      NOP   0;
// --- FCM 01 - Lifting devices ---
      L     "MAL1S032Par".Ilo.ILOMode;
      L     1;
      <>I   ;
      SPB   IO1;
// man on
      U     "MAL1S032Par".Ilo.GrCMDManOn[1];
      S     "G265M".Gr.InManual; // LIFTING DEVICE KILN 1
      R     "MAL1S032Par".Ilo.GrCMDManOn[1];
// man off
      U     "MAL1S032Par".Ilo.GrCMDManOff[1];
      S     "G265M".Gr.CmdManualOff; // LIFTING DEVICE KILN 1
      R     "G265M".Gr.InManual; // LIFTING DEVICE KILN 1
      R     "G265M".USW14; // ILO-cmd
      R     "G265M".USW15; // ILO-cmd
      R     "MAL1S032Par".Ilo.GrCMDManOff[1];
      R     "MAL1S032Par".Ilo.GrCMDManAdditional.Cmd1[1];
      R     "MAL1S032Par".Ilo.GrCMDManAdditional.Cmd2[1];
// man start
      U     "MAL1S032Par".Ilo.GrCMDManStart[1];
      S     "G265M".Gr.CmdOn; // LIFTING DEVICE KILN 1
      S     "G265M".Gr.CmdContinue; // LIFTING DEVICE KILN 1
      R     "MAL1S032Par".Ilo.GrCMDManStart[1];
      U     "MAL1S032Par".Ilo.GrCMDManStart[2];
      R     "MAL1S032Par".Ilo.GrCMDManStart[2];
// man stop
      U     "MAL1S032Par".Ilo.GrCMDManStop[1];
      S     "G265M".Gr.CmdOff; // LIFTING DEVICE KILN 1
      R     "MAL1S032Par".Ilo.GrCMDManStop[1];
// man fault reset
      U     "MAL1S032Par".Ilo.GrCMDManFaultReset[1];
      S     "G265M".Gr.CmdFaultReset; // LIFTING DEVICE KILN 1
      R     "MAL1S032Par".Ilo.GrCMDManFaultReset[1];
// moving direction
      UN    "G265M".Gr.InManual; // LIFTING DEVICE KILN 1
      O(    ;
      L     "MAL1S032Par".Ilo.Code_ILO_Funktion0;
      L     100;
      <>I   ;
      )     ;
      SPB   Stat;
      UN    "MAL1S032Par".Ilo.GrCMDManAdditional.Cmd1[1];
      UN    "MAL1S032Par".Ilo.GrCMDManAdditional.Cmd2[1];
      L     "MAL1S032Par".Par.MachineValue.SOLLWERT_HUBZUG1_HOEHE;
      SPB   Tpos;
      U     "MAL1S032Par".Ilo.GrCMDManAdditional.Cmd1[1]; // ManUp
      L     2000; // 1850mm + Offset = 2000mm
      SPB   Tpos;
      U     "MAL1S032Par".Ilo.GrCMDManAdditional.Cmd2[1]; // ManDown
      L     0; // 0mm
      SPB   Tpos;
      SPA   Stat;
// target position
Tpos: NOP   0;
      T     "MAL1S032Par".Par.ParIntProcess.TarPos_ILO_LiftDev;
Stat: NOP   0;
IO1:  NOP   0;
      NOP   0;
// --- FCM 04 - Fans ---
      L     "MAL1S032Par".Ilo.ILOMode;
      L     4;
      <>I   ;
      SPB   IO4;
// man on
      U     "MAL1S032Par".Ilo.GrCMDManOn[1];
      S     "G271M".Gr.InManual; // FAN KILN 1
//MW 2010.04.06
      S     "G273M".Gr.InManual; // RECYCLING AIR LOUVER KILN 1
      S     "G273M".Gr.CmdOn; // No Button: RECYCLING AIR LOUVER KILN 1
      S     "G273M".Gr.CmdContinue; // No Button RECYCLING AIR LOUVER KILN 1
      R     "MAL1S032Par".Ilo.GrCMDManOn[1];
// man off
      U     "MAL1S032Par".Ilo.GrCMDManOff[1];
      S     "G271M".Gr.CmdManualOff; // FAN KILN 1
      R     "G271M".Gr.InManual; // FAN KILN 1
      R     "G271M".USW14; // ILO-cmd
      R     "G271M".USW15; // ILO-cmd
//MW 2010.04.06
      S     "G273M".Gr.CmdManualOff; // RECYCLING AIR LOUVER KILN 1
      R     "G273M".Gr.InManual; // RECYCLING AIR LOUVER KILN 1
      R     "G273M".USW14; // ILO-cmd
      R     "G273M".USW15; // ILO-cmd
      R     "MAL1S032Par".Ilo.GrCMDManOff[1];
      R     "MAL1S032Par".Ilo.GrCMDManAdditional.Cmd1[1];
      R     "MAL1S032Par".Ilo.GrCMDManAdditional.Cmd2[1];
// man start
      U     "MAL1S032Par".Ilo.GrCMDManStart[1];
      S     "G271M".Gr.CmdOn; // FAN KILN 1
      S     "G271M".Gr.CmdContinue; // FAN KILN 1
//MW 2010.04.06
      S     "G273M".Gr.CmdOn; // No Button: RECYCLING AIR LOUVER KILN 1
      S     "G273M".Gr.CmdContinue; // No Button RECYCLING AIR LOUVER KILN 1
      R     "MAL1S032Par".Ilo.GrCMDManStart[1];
      U     "MAL1S032Par".Ilo.GrCMDManStart[2];
      R     "MAL1S032Par".Ilo.GrCMDManStart[2];
// man stop
      U     "MAL1S032Par".Ilo.GrCMDManStop[1];
      S     "G271M".Gr.CmdOff; // FAN KILN 1
//MW 2010.04.06
//      S     "G273M".Gr.CmdOff           // RECYCLING AIR LOUVER KILN 1
      R     "MAL1S032Par".Ilo.GrCMDManStop[1];
// man fault reset
      U     "MAL1S032Par".Ilo.GrCMDManFaultReset[1];
      S     "G271M".Gr.CmdFaultReset; // FAN KILN 1
//MW 2010.04.06
      S     "G273M".Gr.CmdFaultReset; // RECYCLING AIR LOUVER KILN 1
      R     "MAL1S032Par".Ilo.GrCMDManFaultReset[1];
// target position
      UN    "G271M".Gr.InManual; // FAN KILN 1
      O(    ;
      L     "MAL1S032Par".Ilo.Code_ILO_Funktion0;
      L     400;
      <>I   ;
      )     ;
      SPB   F04a;
      L     "MAL1S032Par".Ilo.SetpointInt01[1];
      T     "MAL1S032Par".Par.ParIntProcess.Speed_ILO_Fan;
F04a: NOP   0;
//MW 2010.04.06
      UN    "G273M".Gr.InManual; // Recycling Air Flap Kilningbox 1
      O(    ;
      L     "MAL1S032Par".Ilo.Code_ILO_Funktion0;
      L     400;
      <>I   ;
      )     ;
      SPB   F04b;
//MW      L     90                          // 90%
      L     100; // 100%
      T     "MAL1S032Par".Par.ParIntProcess.TarPos_ILO_RecycAir;
F04b: NOP   0;

IO4:  NOP   0;
      NOP   0;
// --- FCM 05 - Fans with target air temperature ---
      L     "MAL1S032Par".Ilo.ILOMode;
      L     5;
      <>I   ;
      SPB   IO5;
// man on
      U     "MAL1S032Par".Ilo.GrCMDManOn[1];
      S     "G271M".Gr.InManual; // FAN KILN 1
      S     "G273M".Gr.InManual; // RECYCLING AIR LOUVER KILN 1
      S     "G273M".Gr.CmdOn; // No Button: RECYCLING AIR LOUVER KILN 1
      S     "G273M".Gr.CmdContinue; // No Button RECYCLING AIR LOUVER KILN 1
      S     "G276M".Gr.InManual; // HEATING KILN 1
      S     "G276M".Gr.CmdOn; // No Button: HEATING KILN 1
      S     "G276M".Gr.CmdContinue; // No Button HEATING KILN 1
      S     "G277M".Gr.InManual; // LOUVER AIR HEATER 1 FOR KILN 1
      S     "G277M".Gr.CmdOn; // No Button: LOUVER AIR HEATER 1 FOR KILN 1
      S     "G277M".Gr.CmdContinue; // No Button LOUVER AIR HEATER 1 FOR KILN 1
//MW 2010.04.06      S     "G272M".Gr.InManual         // FRESH AIR LOUVER KILN 1
//MW 2010.04.06      S     "G272M".Gr.CmdOn            // No Button: FRESH AIR LOUVER KILN 1
//MW 2010.04.06      S     "G272M".Gr.CmdContinue      // No Button FRESH AIR LOUVER KILN 1
      S     "G278M".Gr.InManual; // WITHERING AIR KILN 1
      S     "G278M".Gr.CmdOn; // No Button: WITHERING AIR KILN 1
      S     "G278M".Gr.CmdContinue; // No Button WITHERING AIR KILN 1
      R     "MAL1S032Par".Ilo.GrCMDManOn[1];
// man off
      U     "MAL1S032Par".Ilo.GrCMDManOff[1];
      S     "G271M".Gr.CmdManualOff; // FAN KILN 1
      R     "G271M".Gr.InManual; // FAN KILN 1
      R     "G271M".USW14; // ILO-cmd
      R     "G271M".USW15; // ILO-cmd
      S     "G273M".Gr.CmdManualOff; // RECYCLING AIR LOUVER KILN 1
      R     "G273M".Gr.InManual; // RECYCLING AIR LOUVER KILN 1
      R     "G273M".USW14; // ILO-cmd
      R     "G273M".USW15; // ILO-cmd
      S     "G276M".Gr.CmdManualOff; // HEATING KILN 1
      R     "G276M".Gr.InManual; // HEATING KILN 1
      R     "G276M".USW14; // ILO-cmd
      R     "G276M".USW15; // ILO-cmd
      S     "G277M".Gr.CmdManualOff; // LOUVER AIR HEATER 1 FOR KILN 1
      R     "G277M".Gr.InManual; // LOUVER AIR HEATER 1 FOR KILN 1
      R     "G277M".USW14; // ILO-cmd
      R     "G277M".USW15; // ILO-cmd
//MW 2010.04.06      S     "G272M".Gr.CmdManualOff     // FRESH AIR LOUVER KILN 1
//MW 2010.04.06      R     "G272M".Gr.InManual         // FRESH AIR LOUVER KILN 1
      R     "G272M".USW14; // ILO-cmd
      R     "G272M".USW15; // ILO-cmd
      S     "G278M".Gr.CmdManualOff; // WITHERING AIR KILN 1
      R     "G278M".Gr.InManual; // WITHERING AIR KILN 1
      R     "G278M".USW14; // ILO-cmd
      R     "G278M".USW15; // ILO-cmd
      R     "MAL1S032Par".Ilo.GrCMDManOff[1];
      R     "MAL1S032Par".Ilo.GrCMDManAdditional.Cmd1[1];
      R     "MAL1S032Par".Ilo.GrCMDManAdditional.Cmd2[1];
// man start
      U     "MAL1S032Par".Ilo.GrCMDManStart[1];
      S     "G271M".Gr.CmdOn; // FAN KILN 1
      S     "G271M".Gr.CmdContinue; // FAN KILN 1
      S     "G273M".Gr.CmdOn; // RECYCLING AIR LOUVER KILN 1
      S     "G273M".Gr.CmdContinue; // RECYCLING AIR LOUVER KILN 1
      S     "G276M".Gr.CmdOn; // HEATING KILN 1
      S     "G276M".Gr.CmdContinue; // HEATING KILN 1
      S     "G277M".Gr.CmdOn; // LOUVER AIR HEATER 1 FOR KILN 1
      S     "G277M".Gr.CmdContinue; // LOUVER AIR HEATER 1 FOR KILN 1
//MW 2010.04.06      S     "G272M".Gr.CmdOn            // FRESH AIR LOUVER KILN 1
//MW 2010.04.06      S     "G272M".Gr.CmdContinue      // FRESH AIR LOUVER KILN 1
      S     "G278M".Gr.CmdOn; // WITHERING AIR KILN 1
      S     "G278M".Gr.CmdContinue; // WITHERING AIR KILN 1
      R     "MAL1S032Par".Ilo.GrCMDManStart[1];
      U     "MAL1S032Par".Ilo.GrCMDManStart[2];
      R     "MAL1S032Par".Ilo.GrCMDManStart[2];
// man stop
//MW 2010.04.14      U     "MAL1S032Par".Ilo.GrSTMan[17]
      U     "MAL1S032Par".Ilo.GrCMDManStop[1];
      S     "G271M".Gr.CmdOff; // FAN KILN 1
      S     "G273M".Gr.CmdOff; // RECYCLING AIR LOUVER KILN 1
      S     "G276M".Gr.CmdOff; // HEATING KILN 1
      S     "G277M".Gr.CmdOff; // LOUVER AIR HEATER 1 FOR KILN 1
//MW 2010.04.06      S     "G272M".Gr.CmdOff           // FRESH AIR LOUVER KILN 1
      S     "G278M".Gr.CmdOff; // WITHERING AIR KILN 1
//MW 2010.04.14      R     "MAL1S032Par".Ilo.GrSTMan[17]
      R     "MAL1S032Par".Ilo.GrCMDManStop[1];
// man fault reset
      U     "MAL1S032Par".Ilo.GrCMDManFaultReset[1];
      S     "G271M".Gr.CmdFaultReset; // FAN KILN 1
      S     "G273M".Gr.CmdFaultReset; // RECYCLING AIR LOUVER KILN 1
      S     "G276M".Gr.CmdFaultReset; // HEATING KILN 1
      S     "G277M".Gr.CmdFaultReset; // LOUVER AIR HEATER 1 FOR KILN 1
//MW 2010.04.06      S     "G272M".Gr.CmdFaultReset    // FRESH AIR LOUVER KILN 1
      S     "G278M".Gr.CmdFaultReset; // WITHERING AIR KILN 1
      R     "MAL1S032Par".Ilo.GrCMDManFaultReset[1];
// target position
      UN    "G271M".Gr.InManual; // FAN KILN 1
      O(    ;
      L     "MAL1S032Par".Ilo.Code_ILO_Funktion0;
      L     500;
      <>I   ;
      )     ;
      SPB   F05b;
      L     "MAL1S032Par".Ilo.SetpointInt01[1];
      T     "MAL1S032Par".Par.ParIntProcess.Speed_ILO_Fan;
F05b: NOP   0;
      UN    "G273M".Gr.InManual; // Recycling Air Flap Kilningbox 1
      O(    ;
      L     "MAL1S032Par".Ilo.Code_ILO_Funktion0;
      L     500;
      <>I   ;
      )     ;
      SPB   F05c;
      L     "MAL1S032Par".Ilo.SetpointInt03[1];
      T     "MAL1S032Par".Par.ParIntProcess.TarPos_ILO_RecycAir;
F05c: NOP   0;
      UN    "G278M".Gr.InManual; // Withering Air Flap Kilningbox 1
      O(    ;
      L     "MAL1S032Par".Ilo.Code_ILO_Funktion0;
      L     500;
      <>I   ;
      )     ;
      SPB   F05d;
      L     "MAL1S032Par".Ilo.SetpointInt04[1];
      T     "MAL1S032Par".Par.ParIntProcess.TarPos_ILO_WitheringAir;
F05d: NOP   0;
      UN    "G276M".Gr.InManual; // Heating Kiln 1
      O(    ;
      L     "MAL1S032Par".Ilo.Code_ILO_Funktion0;
      L     500;
      <>I   ;
      )     ;
      SPB   F05e;
//MW 2010.04.06      L     "MAL1S032Par".Ilo.SetpointInt01[2]
      L     "MAL1S032Par".Ilo.SetpointInt02[1];
      T     "MAL1S032Par".Par.ParIntProcess.TargetTemperature_ILO;
F05e: NOP   0;

IO5:  NOP   0;
      NOP   0;
// --- FCM 06 - Fresh air flap ---
      L     "MAL1S032Par".Ilo.ILOMode;
      L     6;
      <>I   ;
      SPB   IO6;
// man on
      U     "MAL1S032Par".Ilo.GrCMDManOn[1];
      S     "G272M".Gr.InManual; // FRESH AIR LOUVER KILN 1
      R     "MAL1S032Par".Ilo.GrCMDManOn[1];
// man off
      U     "MAL1S032Par".Ilo.GrCMDManOff[1];
      S     "G272M".Gr.CmdManualOff; // FRESH AIR LOUVER KILN 1
      R     "G272M".Gr.InManual; // FRESH AIR LOUVER KILN 1
      R     "G272M".USW14; // ILO-cmd
      R     "G272M".USW15; // ILO-cmd
      R     "MAL1S032Par".Ilo.GrCMDManOff[1];
      R     "MAL1S032Par".Ilo.GrCMDManAdditional.Cmd1[1];
      R     "MAL1S032Par".Ilo.GrCMDManAdditional.Cmd2[1];
// man start
      U     "MAL1S032Par".Ilo.GrCMDManStart[1];
      S     "G272M".Gr.CmdOn; // FRESH AIR LOUVER KILN 1
      S     "G272M".Gr.CmdContinue; // FRESH AIR LOUVER KILN 1
      R     "MAL1S032Par".Ilo.GrCMDManStart[1];
      U     "MAL1S032Par".Ilo.GrCMDManStart[2];
      R     "MAL1S032Par".Ilo.GrCMDManStart[2];
// man stop
      U     "MAL1S032Par".Ilo.GrCMDManStop[1];
      S     "G272M".Gr.CmdOff; // FRESH AIR LOUVER KILN 1
      R     "MAL1S032Par".Ilo.GrCMDManStop[1];
// man fault reset
      U     "MAL1S032Par".Ilo.GrCMDManFaultReset[1];
      S     "G272M".Gr.CmdFaultReset; // FRESH AIR LOUVER KILN 1
      R     "MAL1S032Par".Ilo.GrCMDManFaultReset[1];
// moving direction

// target position
      UN    "G272M".Gr.InManual; // FRESH AIR LOUVER KILN 1
      SPB   F06b;
      L     "MAL1S032Par".Ilo.SetpointInt01[1];
      T     "MAL1S032Par".Par.ParIntProcess.TarPos_ILO_FreshAir;
F06b: NOP   0;

IO6:  NOP   0;
      NOP   0;
// --- FCM 07 - Recycling air flap ---
      L     "MAL1S032Par".Ilo.ILOMode;
      L     7;
      <>I   ;
      SPB   IO7;
// man on
      U     "MAL1S032Par".Ilo.GrCMDManOn[1];
      S     "G273M".Gr.InManual; // RECYCLING AIR LOUVER KILN 1
      S     "G278M".Gr.InManual; // WITHERING AIR KILN 1
      R     "MAL1S032Par".Ilo.GrCMDManOn[1];
// man off
      U     "MAL1S032Par".Ilo.GrCMDManOff[1];
      S     "G273M".Gr.CmdManualOff; // RECYCLING AIR LOUVER KILN 1
      R     "G273M".Gr.InManual; // RECYCLING AIR LOUVER KILN 1
      R     "G273M".USW14; // ILO-cmd
      R     "G273M".USW15; // ILO-cmd
      S     "G278M".Gr.CmdManualOff; // WITHERING AIR KILN 1
      R     "G278M".Gr.InManual; // WITHERING AIR KILN 1
      R     "G278M".USW14; // ILO-cmd
      R     "G278M".USW15; // ILO-cmd
      R     "MAL1S032Par".Ilo.GrCMDManOff[1];
      R     "MAL1S032Par".Ilo.GrCMDManAdditional.Cmd1[1];
      R     "MAL1S032Par".Ilo.GrCMDManAdditional.Cmd2[1];
// man start
      U     "MAL1S032Par".Ilo.GrCMDManStart[1];
      S     "G273M".Gr.CmdOn; // RECYCLING AIR LOUVER KILN 1
      S     "G273M".Gr.CmdContinue; // RECYCLING AIR LOUVER KILN 1
      S     "G278M".Gr.CmdOn; // WITHERING AIR KILN 1
      S     "G278M".Gr.CmdContinue; // WITHERING AIR KILN 1
      R     "MAL1S032Par".Ilo.GrCMDManStart[1];
      U     "MAL1S032Par".Ilo.GrCMDManStart[2];
      R     "MAL1S032Par".Ilo.GrCMDManStart[2];
// man stop
      U     "MAL1S032Par".Ilo.GrCMDManStop[1];
      S     "G273M".Gr.CmdOff; // RECYCLING AIR LOUVER KILN 1
      S     "G278M".Gr.CmdOff; // WITHERING AIR KILN 1
      R     "MAL1S032Par".Ilo.GrCMDManStop[1];
// man fault reset
      U     "MAL1S032Par".Ilo.GrCMDManFaultReset[1];
      S     "G273M".Gr.CmdFaultReset; // RECYCLING AIR LOUVER KILN 1
      S     "G278M".Gr.CmdFaultReset; // WITHERING AIR KILN 1
      R     "MAL1S032Par".Ilo.GrCMDManFaultReset[1];
// moving direction

// target position
      UN    "G273M".Gr.InManual; // RECYCLING AIR LOUVER KILN 1
      SPB   F07a;
      L     "MAL1S032Par".Ilo.SetpointInt01[1];
      T     "MAL1S032Par".Par.ParIntProcess.TarPos_ILO_RecycAir;
F07a: NOP   0;
IO7:  NOP   0;
      NOP   0;
// --- FCM 09 - Floor drives ---
      L     "MAL1S032Par".Ilo.ILOMode;
      L     9;
      <>I   ;
      SPB   IO9;
// man on
      U     "MAL1S032Par".Ilo.GrCMDManOn[1];
      S     "G266M".Gr.InManual; // TRAVELLING DRIVE KILN 1
      R     "MAL1S032Par".Ilo.GrCMDManOn[1];
// man off
      U     "MAL1S032Par".Ilo.GrCMDManOff[1];
      S     "G266M".Gr.CmdManualOff; // TRAVELLING DRIVE KILN 1
      R     "G266M".Gr.InManual; // TRAVELLING DRIVE KILN 1
      R     "G266M".USW14; // ILO-cmd
      R     "G266M".USW15; // ILO-cmd
      R     "MAL1S032Par".Ilo.GrCMDManOff[1];
      R     "MAL1S032Par".Ilo.GrCMDManAdditional.Cmd1[1];
      R     "MAL1S032Par".Ilo.GrCMDManAdditional.Cmd2[1];
// man start
      U     "MAL1S032Par".Ilo.GrCMDManStart[1];
      S     "G266M".Gr.CmdOn; // TRAVELLING DRIVE KILN 1
      S     "G266M".Gr.CmdContinue; // TRAVELLING DRIVE KILN 1
      R     "MAL1S032Par".Ilo.GrCMDManStart[1];
      U     "MAL1S032Par".Ilo.GrCMDManStart[2];
      R     "MAL1S032Par".Ilo.GrCMDManStart[2];
// man stop
      U     "MAL1S032Par".Ilo.GrCMDManStop[1];
      S     "G266M".Gr.CmdOff; // TRAVELLING DRIVE KILN 1
      R     "MAL1S032Par".Ilo.GrCMDManStop[1];
// man fault reset
      U     "MAL1S032Par".Ilo.GrCMDManFaultReset[1];
      S     "G266M".Gr.CmdFaultReset; // TRAVELLING DRIVE KILN 1
      R     "MAL1S032Par".Ilo.GrCMDManFaultReset[1];
      NOP   0;
      UN    "G266M".Gr.InManual; // TRAVELLING DRIVE KILN 1
      O     ;
      UN    "MAL1S032Par".Ilo.GrCMDManAdditional.Cmd1[1];
      UN    "MAL1S032Par".Ilo.GrCMDManAdditional.Cmd2[1];
      SPB   f092;
      U     "MAL1S032Par".Ilo.GrCMDManAdditional.Cmd1[1];
      =     "G266M".USW14; // ILO-cmd run fwd
      U     "MAL1S032Par".Ilo.GrCMDManAdditional.Cmd2[1];
      =     "G266M".USW15; // ILO-cmd run rev
// target position
      L     "MAL1S032Par".Ilo.SetpointInt01[1];
      T     "MAL1S032Par".Par.ParIntProcess.Speed_ILO_FloorRotating;
f092: NOP   0;

IO9:  NOP   0;
      NOP   0;
// --- FCM 10 - Floor drives and lifting devices ---
      L     "MAL1S032Par".Ilo.ILOMode;
      L     10;
      <>I   ;
      SPB   IO10;
// man on
      U     "MAL1S032Par".Ilo.GrCMDManOn[1];
      S     "G265M".Gr.InManual; // LIFTING DEVICE KILN 1
      S     "G265M".Gr.CmdOn; // No Button: LIFTING DEVICE KILN 1
      S     "G265M".Gr.CmdContinue; // No Button LIFTING DEVICE KILN 1
      S     "G266M".Gr.InManual; // TRAVELLING DRIVE KILN 1
      R     "MAL1S032Par".Ilo.GrCMDManOn[1];
// man off
      U     "MAL1S032Par".Ilo.GrCMDManOff[1];
      S     "G265M".Gr.CmdManualOff; // LIFTING DEVICE KILN 1
      R     "G265M".Gr.InManual; // LIFTING DEVICE KILN 1
      R     "G265M".USW14; // ILO-cmd
      R     "G265M".USW15; // ILO-cmd
      S     "G266M".Gr.CmdManualOff; // TRAVELLING DRIVE KILN 1
      R     "G266M".Gr.InManual; // TRAVELLING DRIVE KILN 1
      R     "G266M".USW14; // ILO-cmd
      R     "G266M".USW15; // ILO-cmd
      R     "MAL1S032Par".Ilo.GrCMDManOff[1];
      R     "MAL1S032Par".Ilo.GrCMDManAdditional.Cmd1[1];
      R     "MAL1S032Par".Ilo.GrCMDManAdditional.Cmd2[1];
// man start
      U     "MAL1S032Par".Ilo.GrCMDManStart[1];
      S     "G266M".Gr.CmdOn; // TRAVELLING DRIVE KILN 1
      S     "G266M".Gr.CmdContinue; // TRAVELLING DRIVE KILN 1
      R     "MAL1S032Par".Ilo.GrCMDManStart[1];
      U     "MAL1S032Par".Ilo.GrCMDManStart[2];
      S     "G265M".Gr.CmdOn; // LIFTING DEVICE KILN 1
      S     "G265M".Gr.CmdContinue; // LIFTING DEVICE KILN 1
      R     "MAL1S032Par".Ilo.GrCMDManStart[2];
      U     "MAL1S032Par".Ilo.GrCMDManStart[3];
      R     "MAL1S032Par".Ilo.GrCMDManStart[3];
// man stop
      U     "MAL1S032Par".Ilo.GrCMDManStop[1];
      S     "G265M".Gr.CmdOff; // LIFTING DEVICE KILN 1
      S     "G266M".Gr.CmdOff; // TRAVELLING DRIVE KILN 1
      R     "MAL1S032Par".Ilo.GrCMDManStop[1];
// man fault reset
      U     "MAL1S032Par".Ilo.GrCMDManFaultReset[1];
      S     "G265M".Gr.CmdFaultReset; // LIFTING DEVICE KILN 1
      S     "G266M".Gr.CmdFaultReset; // TRAVELLING DRIVE KILN 1
      R     "MAL1S032Par".Ilo.GrCMDManFaultReset[1];
// moving direction
      NOP   0;
      UN    "G266M".Gr.InManual; // TRAVELLING DRIVE KILN 1
      O     ;
      UN    "MAL1S032Par".Ilo.GrCMDManAdditional.Cmd1[1];
      UN    "MAL1S032Par".Ilo.GrCMDManAdditional.Cmd2[1];
      SPB   f102;
      U     "MAL1S032Par".Ilo.GrCMDManAdditional.Cmd1[1];
      =     "G266M".USW14; // ILO-cmd run fwd
      U     "MAL1S032Par".Ilo.GrCMDManAdditional.Cmd2[1];
      =     "G266M".USW15; // ILO-cmd run rev
// target speed floor drives
      L     "MAL1S032Par".Ilo.SetpointInt01[1];
      T     "MAL1S032Par".Par.ParIntProcess.Speed_ILO_FloorRotating;
f102: NOP   0;
      UN    "G265M".Gr.InManual; // LIFTING DEVICE KILN 1
      O(    ;
      L     "MAL1S032Par".Ilo.Code_ILO_Funktion0;
      L     1000;
      <>I   ;
      )     ;
      SPB   f103;
// target position lifting devices
      L     "MAL1S032Par".Ilo.SetpointInt02[1];
      T     "MAL1S032Par".Par.ParIntProcess.TarPos_ILO_LiftDev;
f103: NOP   0;

IO10: NOP   0;
      NOP   0;
// --- FCM 11 - Floor drives and lifting devices and screw ---
      L     "MAL1S032Par".Ilo.ILOMode;
      L     11;
      <>I   ;
      SPB   IO11;
// man on
      U     "MAL1S032Par".Ilo.GrCMDManOn[1];
      S     "G265M".Gr.InManual; // LIFTING DEVICE KILN 1
      S     "G265M".Gr.CmdOn; // No Button: LIFTING DEVICE KILN 1
      S     "G265M".Gr.CmdContinue; // No Button LIFTING DEVICE KILN 1
      S     "G266M".Gr.InManual; // TRAVELLING DRIVE KILN 1
      S     "G267M".Gr.InManual; // UNLOADING / LOADING SCREW KILN 1
      R     "MAL1S032Par".Ilo.GrCMDManOn[1];
// man off
      U     "MAL1S032Par".Ilo.GrCMDManOff[1];
      S     "G265M".Gr.CmdManualOff; // LIFTING DEVICE KILN 1
      R     "G265M".Gr.InManual; // LIFTING DEVICE KILN 1
      R     "G265M".USW14; // ILO-cmd
      R     "G265M".USW15; // ILO-cmd
      S     "G266M".Gr.CmdManualOff; // TRAVELLING DRIVE KILN 1
      R     "G266M".Gr.InManual; // TRAVELLING DRIVE KILN 1
      R     "G266M".USW14; // ILO-cmd
      R     "G266M".USW15; // ILO-cmd
      S     "G267M".Gr.CmdManualOff; // UNLOADING / LOADING SCREW KILN 1
      R     "G267M".Gr.InManual; // UNLOADING / LOADING SCREW KILN 1
      R     "G267M".USW14; // ILO-cmd
      R     "G267M".USW15; // ILO-cmd
      R     "MAL1S032Par".Ilo.GrCMDManOff[1];
      R     "MAL1S032Par".Ilo.GrCMDManAdditional.Cmd1[1];
      R     "MAL1S032Par".Ilo.GrCMDManAdditional.Cmd2[1];
// man start
      U     "MAL1S032Par".Ilo.GrCMDManStart[1];
      S     "G266M".Gr.CmdOn; // TRAVELLING DRIVE KILN 1
      S     "G266M".Gr.CmdContinue; // TRAVELLING DRIVE KILN 1
      R     "MAL1S032Par".Ilo.GrCMDManStart[1];
      U     "MAL1S032Par".Ilo.GrCMDManStart[2];
      S     "G265M".Gr.CmdOn; // LIFTING DEVICE KILN 1
      S     "G265M".Gr.CmdContinue; // LIFTING DEVICE KILN 1
      R     "MAL1S032Par".Ilo.GrCMDManStart[2];
      U     "MAL1S032Par".Ilo.GrCMDManStart[3];
      S     "G267M".Gr.CmdOn; // UNLOADING / LOADING SCREW KILN 1
      S     "G267M".Gr.CmdContinue; // UNLOADING / LOADING SCREW KILN 1
      R     "MAL1S032Par".Ilo.GrCMDManStart[3];
//MW      U     "MAL1S032Par".Ilo.GrCMDManStart[4]
//MW      S     "G267M".Gr.CmdOn            // UNLOADING / LOADING SCREW KILN 1
//MW      S     "G267M".Gr.CmdContinue      // UNLOADING / LOADING SCREW KILN 1
//MW      R     "MAL1S032Par".Ilo.GrCMDManStart[4]
// man stop
      U     "MAL1S032Par".Ilo.GrCMDManStop[1];
      S     "G265M".Gr.CmdOff; // LIFTING DEVICE KILN 1
      S     "G266M".Gr.CmdOff; // TRAVELLING DRIVE KILN 1
      S     "G267M".Gr.CmdOff; // UNLOADING / LOADING SCREW KILN 1
      R     "MAL1S032Par".Ilo.GrCMDManStop[1];
// man fault reset
      U     "MAL1S032Par".Ilo.GrCMDManFaultReset[1];
      S     "G265M".Gr.CmdFaultReset; // LIFTING DEVICE KILN 1
      S     "G266M".Gr.CmdFaultReset; // TRAVELLING DRIVE KILN 1
      S     "G267M".Gr.CmdFaultReset; // UNLOADING / LOADING SCREW KILN 1
      R     "MAL1S032Par".Ilo.GrCMDManFaultReset[1];
// moving direction
      UN    "G266M".Gr.InManual; // TRAVELLING DRIVE KILN 1
      O     ;
      UN    "MAL1S032Par".Ilo.GrCMDManAdditional.Cmd1[1];
      UN    "MAL1S032Par".Ilo.GrCMDManAdditional.Cmd2[1];
      SPB   f112;
      U     "MAL1S032Par".Ilo.GrCMDManAdditional.Cmd1[1];
      =     "G266M".USW14; // ILO-cmd run fwd
      U     "MAL1S032Par".Ilo.GrCMDManAdditional.Cmd2[1];
      =     "G266M".USW15; // ILO-cmd run rev
// target speed floor drives
      L     "MAL1S032Par".Ilo.SetpointInt01[1];
      T     "MAL1S032Par".Par.ParIntProcess.Speed_ILO_FloorRotating;
f112: NOP   0;
      UN    "G265M".Gr.InManual; // Malting Plant OAO Belsolod Ivanonvo Weissrussland
      O(    ;
      L     "MAL1S032Par".Ilo.Code_ILO_Funktion0;
      L     1100;
      <>I   ;
      )     ;
      SPB   f113;
// target position lifting devices
      L     "MAL1S032Par".Ilo.SetpointInt01[2];
      L     "MAL1S032Par".Ilo.SetpointInt02[1];
      T     "MAL1S032Par".Par.ParIntProcess.TarPos_ILO_LiftDev;
f113: NOP   0;
      UN    "G267M".Gr.InManual; // UNLOADING / LOADING SCREW KILN 1
      O     ;
      UN    "MAL1S032Par".Ilo.GrCMDManAdditional.Cmd1[3];
      UN    "MAL1S032Par".Ilo.GrCMDManAdditional.Cmd2[3];
      SPB   f114;
      U     "MAL1S032Par".Ilo.GrCMDManAdditional.Cmd1[3];
      =     "G267M".USW14; // ILO-cmd run fwd
      U     "MAL1S032Par".Ilo.GrCMDManAdditional.Cmd2[3];
      =     "G267M".USW15; // ILO-cmd run rev
f114: NOP   0;
IO11: NOP   0;
      NOP   0;
// --- FCM 12 - Floor drives and lifting devices and screw and discharging flap ---
      L     "MAL1S032Par".Ilo.ILOMode;
      L     12;
      <>I   ;
      SPB   IO12;
// man on
      U     "MAL1S032Par".Ilo.GrCMDManOn[1];
      S     "G265M".Gr.InManual; // LIFTING DEVICE KILN 1
      S     "G265M".Gr.CmdOn; // No Button: LIFTING DEVICE KILN 1
      S     "G265M".Gr.CmdContinue; // No Button LIFTING DEVICE KILN 1
      S     "G266M".Gr.InManual; // TRAVELLING DRIVE KILN 1
      S     "G267M".Gr.InManual; // UNLOADING / LOADING SCREW KILN 1
      S     "G268M".Gr.InManual; // DISCHARGE DOOR KILN 1
      R     "MAL1S032Par".Ilo.GrCMDManOn[1];
// man off
      U     "MAL1S032Par".Ilo.GrCMDManOff[1];
      S     "G265M".Gr.CmdManualOff; // LIFTING DEVICE KILN 1
      R     "G265M".Gr.InManual; // LIFTING DEVICE KILN 1
      R     "G265M".USW14; // ILO-cmd
      R     "G265M".USW15; // ILO-cmd
      S     "G266M".Gr.CmdManualOff; // TRAVELLING DRIVE KILN 1
      R     "G266M".Gr.InManual; // TRAVELLING DRIVE KILN 1
      R     "G266M".USW14; // ILO-cmd
      R     "G266M".USW15; // ILO-cmd
      S     "G267M".Gr.CmdManualOff; // UNLOADING / LOADING SCREW KILN 1
      R     "G267M".Gr.InManual; // UNLOADING / LOADING SCREW KILN 1
      R     "G267M".USW14; // ILO-cmd
      R     "G267M".USW15; // ILO-cmd
      S     "G268M".Gr.CmdManualOff; // DISCHARGE DOOR KILN 1
      R     "G268M".Gr.InManual; // DISCHARGE DOOR KILN 1
      R     "G268M".USW14; // ILO-cmd
      R     "G268M".USW15; // ILO-cmd
      R     "MAL1S032Par".Ilo.GrCMDManOff[1];
      R     "MAL1S032Par".Ilo.GrCMDManAdditional.Cmd1[1];
      R     "MAL1S032Par".Ilo.GrCMDManAdditional.Cmd2[1];
// man start
      U     "MAL1S032Par".Ilo.GrCMDManStart[1];
      S     "G266M".Gr.CmdOn; // TRAVELLING DRIVE KILN 1
      S     "G266M".Gr.CmdContinue; // TRAVELLING DRIVE KILN 1
      R     "MAL1S032Par".Ilo.GrCMDManStart[1];
      U     "MAL1S032Par".Ilo.GrCMDManStart[2];
      S     "G265M".Gr.CmdOn; // LIFTING DEVICE KILN 1
      S     "G265M".Gr.CmdContinue; // LIFTING DEVICE KILN 1
      R     "MAL1S032Par".Ilo.GrCMDManStart[2];
      U     "MAL1S032Par".Ilo.GrCMDManStart[3];
      S     "G267M".Gr.CmdOn; // UNLOADING / LOADING SCREW KILN 1
      S     "G267M".Gr.CmdContinue; // UNLOADING / LOADING SCREW KILN 1
      R     "MAL1S032Par".Ilo.GrCMDManStart[3];
      U     "MAL1S032Par".Ilo.GrCMDManStart[4];
//MW 2010.04.16      S     "G267M".Gr.CmdOn            // UNLOADING / LOADING SCREW KILN 1
//MW 2010.04.16      S     "G267M".Gr.CmdContinue      // UNLOADING / LOADING SCREW KILN 1
      S     "G268M".Gr.CmdOn; // DISCHARGE DOOR KILN 1
      S     "G268M".Gr.CmdContinue; // DISCHARGE DOOR KILN 1
      R     "MAL1S032Par".Ilo.GrCMDManStart[4];
// man stop
      U     "MAL1S032Par".Ilo.GrCMDManStop[1];
      S     "G265M".Gr.CmdOff; // LIFTING DEVICE KILN 1
      S     "G266M".Gr.CmdOff; // TRAVELLING DRIVE KILN 1
      S     "G267M".Gr.CmdOff; // UNLOADING / LOADING SCREW KILN 1
      S     "G268M".Gr.CmdOff; // DISCHARGE DOOR KILN 1
      R     "MAL1S032Par".Ilo.GrCMDManStop[1];
// man fault reset
      U     "MAL1S032Par".Ilo.GrCMDManFaultReset[1];
      S     "G265M".Gr.CmdFaultReset; // LIFTING DEVICE KILN 1
      S     "G266M".Gr.CmdFaultReset; // TRAVELLING DRIVE KILN 1
      S     "G267M".Gr.CmdFaultReset; // UNLOADING / LOADING SCREW KILN 1
      S     "G268M".Gr.CmdFaultReset; // DISCHARGE DOOR KILN 1
      R     "MAL1S032Par".Ilo.GrCMDManFaultReset[1];
// moving direction
      UN    "G266M".Gr.InManual; // TRAVELLING DRIVE KILN 1
      O     ;
      UN    "MAL1S032Par".Ilo.GrCMDManAdditional.Cmd1[1];
      UN    "MAL1S032Par".Ilo.GrCMDManAdditional.Cmd2[1];
      SPB   f122;
      U     "MAL1S032Par".Ilo.GrCMDManAdditional.Cmd1[1];
      =     "G266M".USW14; // ILO-cmd run fwd
      U     "MAL1S032Par".Ilo.GrCMDManAdditional.Cmd2[1];
      =     "G266M".USW15; // ILO-cmd run rev
// target speed floor drives
      L     "MAL1S032Par".Ilo.SetpointInt01[1];
      T     "MAL1S032Par".Par.ParIntProcess.Speed_ILO_FloorRotating;
f122: NOP   0;
      UN    "G265M".Gr.InManual; // LIFTING DEVICE KILN 1
      O(    ;
      L     "MAL1S032Par".Ilo.Code_ILO_Funktion0;
      L     1200;
      <>I   ;
      )     ;
      SPB   f123;
// target position lifting devices
      L     "MAL1S032Par".Ilo.SetpointInt02[1];
      T     "MAL1S032Par".Par.ParIntProcess.TarPos_ILO_LiftDev;
f123: NOP   0;
      UN    "G267M".Gr.InManual; // Malting Plant OAO Belsolod Ivanonvo Weissrussland
      O     ;
      UN    "MAL1S032Par".Ilo.GrCMDManAdditional.Cmd1[3];
      UN    "MAL1S032Par".Ilo.GrCMDManAdditional.Cmd2[3];
      SPB   f124;
      U     "MAL1S032Par".Ilo.GrCMDManAdditional.Cmd1[3];
//JV070810      =     "G267M".USW14               // ILO-cmd run fwd
      =     "G267M".USW15; // ILO-cmd run rev  //JV070810 nur entladen
      R     "G267M".USW14; // ILO-cmd run fwd  //JV070810 nur entladen
      U     "MAL1S032Par".Ilo.GrCMDManAdditional.Cmd2[3];
      =     "G267M".USW15; // ILO-cmd run rev  //JV070810 nur entladen
      R     "G267M".USW14; // ILO-cmd run fwd  //JV070810 nur entladen

f124: NOP   0;
      UN    "G268M".Gr.InManual; // DISCHARGE DOOR KILN 1
      O     ;
      UN    "MAL1S032Par".Ilo.GrCMDManAdditional.Cmd1[4];
      UN    "MAL1S032Par".Ilo.GrCMDManAdditional.Cmd2[4];
      SPB   f125;
      U     "MAL1S032Par".Ilo.GrCMDManAdditional.Cmd1[4];
      =     "G268M".USW14; // ILO-cmd OPEN
      U     "MAL1S032Par".Ilo.GrCMDManAdditional.Cmd2[4];
      =     "G268M".USW15; // ILO-cmd CLOSE
f125: NOP   0;
IO12: NOP   0;
//
// copy state
      U     "G265M".Gr.InOutAutostartMan; // LIFTING DEVICE KILN 1
      =     "MAL1S032Par".Ilo.GrSTMan[1];
      U     "G266M".Gr.InOutAutostartMan; // TRAVELLING DRIVE KILN 1
      =     "MAL1S032Par".Ilo.GrSTMan[2];
      U     "G267M".Gr.InOutAutostartMan; // UNLOADING / LOADING SCREW KILN 1
      =     "MAL1S032Par".Ilo.GrSTMan[3];
      U     "G268M".Gr.InOutAutostartMan; // DISCHARGE DOOR KILN 1
      =     "MAL1S032Par".Ilo.GrSTMan[4];
      U     "G271M".Gr.InOutAutostartMan; // FAN KILN 1
      =     "MAL1S032Par".Ilo.GrSTMan[6];
      U     "G276M".Gr.InOutAutostartMan; // HEATING KILN 1
      =     "MAL1S032Par".Ilo.GrSTMan[11];
      U     "G277M".Gr.InOutAutostartMan; // LOUVER AIR HEATER 1 FOR KILN 1
      =     "MAL1S032Par".Ilo.GrSTMan[12];
      U     "G272M".Gr.InOutAutostartMan; // FRESH AIR LOUVER KILN 1
      =     "MAL1S032Par".Ilo.GrSTMan[13];
      U     "G278M".Gr.InOutAutostartMan; // WITHERING AIR KILN 1
      =     "MAL1S032Par".Ilo.GrSTMan[14];
      U     "G273M".Gr.InOutAutostartMan; // RECYCLING AIR LOUVER KILN 1
      =     "MAL1S032Par".Ilo.GrSTMan[15];
      U     "G279M".Gr.InOutAutostartMan; // HEATING KILN 1 + 2
      =     "MAL1S032Par".Ilo.GrSTMan[16];
NETWORK
TITLE =ASW_9999: Init Flag
// clear all flags explicde to find them back
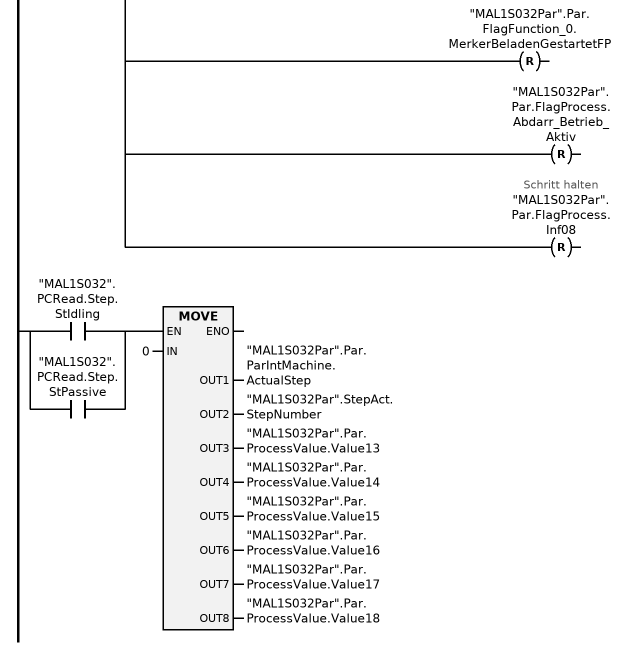
      U     "MAL1S032".PCRead.Step.StIdling;
      O     "MAL1S032".PCRead.Step.StPassive;
      R     "MAL1S032Par".Par.FlagFunction_1.StepLoading;
      R     "MAL1S032Par".Par.FlagFunction_1.StepUnloading;
      R     "MAL1S032Par".Par.FlagFunction_1.StepCleaning;
      R     "MAL1S032Par".Par.FlagFunction_1.LoadingBreak;
      R     "MAL1S032Par".Par.FlagFunction_1.UnloadingBreak;
      R     "MAL1S032Par".Par.FlagFunction_1.CleaningBreak;
      R     "MAL1S032Par".Par.FlagFunction_1.FinishLoading;
      R     "MAL1S032Par".Par.FlagFunction_1.FinishUnloading;
      R     "MAL1S032Par".Par.FlagFunction_1.FinishCleaning;
      R     "MAL1S032Par".Par.FlagFunction_1.Entladerunden_erreicht;
      R     "MAL1S032Par".Par.FlagFunction_1.Reinigungsrunde_erreicht;
      R     "MAL1S032Par".Par.FlagFunction_1.UnloadEnd;
      R     "MAL1S032Par".Par.FlagFunction_1.LoadEnd;
      R     "MAL1S032Par".Par.FlagFunction_1.UnloadFirstPart;
      R     "MAL1S032Par".Par.FlagFunction_1.UnloadSecondPart;
      R     "MAL1S032Par".Par.FlagProcess.ProcessActive;
      R     "MAL1S032Par".Par.FlagProcess.StartProzess_FP;
      R     "MAL1S032Par".Par.FlagProcess.StartProzess_SCAN;
      R     "MAL1S032Par".Par.FlagProcess.TurningFloor;
      R     "MAL1S032Par".Par.FlagProcess.Cooling_Activ;
      R     "MAL1S032Par".Par.FlagProcess.FP_SendResultToPIC;
      R     "MAL1S032Par".Par.FlagProcess.ProcessEnd;

// --> Wie bei Bank Avangard
//MW 2010.04.06
      U     "MAL1S032".PCRead.Step.StPassive;
      R     "MAL1S032Par".Par.FlagMachine.WEGMESSUNG_0_FLAG;
      R     "MAL1S032Par".Par.FlagMachine.ImpulsNullstellung;
      R     "MAL1S032Par".Par.FlagMachine.CmdTurnFwdAfterLoading;
      R     "MAL1S032Par".Par.FlagMachine.CmdTurnRevAfterLoading;
      R     "MAL1S032Par".Par.FlagMachine.ImpulsNullstellungFP;
      R     "MAL1S032Par".Par.FlagMachine.CmdTurnFwdAfterTurning;
      R     "MAL1S032Par".Par.FlagMachine.CmdTurnRevAfterTurning;
      R     "MAL1S032Par".Par.FlagMachine.WEGMESSUNG_0;
      R     "MAL1S032Par".Par.FlagMachine.CmdTurnFwdAfterUnloading;
      R     "MAL1S032Par".Par.FlagMachine.CmdTurnRevAfterUnloading;
      R     "MAL1S032Par".Par.FlagMachine.NULL_INDEX_FP;
      R     "MAL1S032Par".Par.FlagFunction_0.MerkerBeladenGestartetFP;
      R     "MAL1S032Par".Par.FlagProcess.Abdarr_Betrieb_Aktiv;
      R     "MAL1S032Par".Par.FlagProcess.Inf08; // Schritt halten
//
      U     "MAL1S032".PCRead.Step.StIdling;
      O     "MAL1S032".PCRead.Step.StPassive;
      SPBN  csn;
      L     0; // clear step number
      T     "MAL1S032Par".Par.ParIntMachine.ActualStep;
      T     "MAL1S032Par".StepAct.StepNumber;
      T     "MAL1S032Par".Par.ProcessValue.Value13; // Schaltpunkt Regelung
      T     "MAL1S032Par".Par.ProcessValue.Value14; // Sollwert Umluftklappen Kühlen
      T     "MAL1S032Par".Par.ProcessValue.Value15; // Sollwert Ventilator Kühlen
      T     "MAL1S032Par".Par.ProcessValue.Value16; // Step Copy
      T     "MAL1S032Par".Par.ProcessValue.Value17; // Sollwert Umluftklappen Kühlen
      T     "MAL1S032Par".Par.ProcessValue.Value18; // Sollwert Ventilator Kühlen

csn:  NOP   0;

NETWORK
TITLE =Main0_End: Init flag
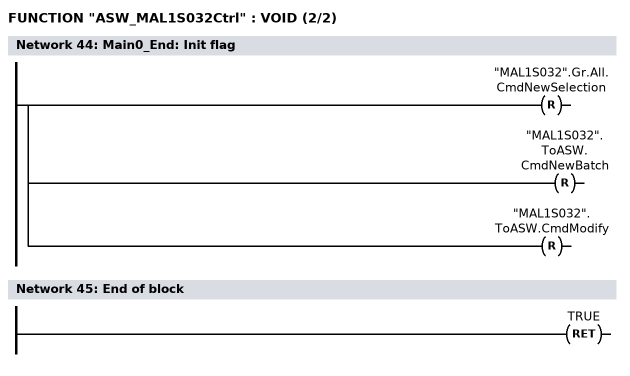

      SET   ;
      R     "MAL1S032".Gr.All.CmdNewSelection;
      R     "MAL1S032".ToASW.CmdNewBatch;
      R     "MAL1S032".ToASW.CmdModify;

NETWORK
TITLE =End of block

      BE    ;

END_FUNCTION

